PROGRAM Ignition
VAR
END_VAR
VAR_OUTPUT
	err : UINT;
END_VAR

// check that no error is occuring
IF (GVL.nError <> ErrorCode.SUCCESS) THEN
	err := GVL.nError;
RETURN;
END_IF

// flame detect

// start iginition
// clean gases

END_PROGRAM

(* stored: Version 1.1.0.1, ProductVersion 3.1.4022.18
   POU Ignition: Id {fa1eb9f1-d6d2-4838-8fbb-7ff8260d154b}, SpecialFunc None *)
